FUNCTION TryConvert_REAL_TO_UINT : BOOL
VAR_INPUT
	in : REAL;
	out : REFERENCE TO UINT;
END_VAR

IF in > DatatypeLimits.MAX_VALUE_OF_REAL_WHICH_CAN_BE_HELD_IN_A_UINT THEN
	RETURN;
END_IF

IF in < DatatypeLimits.MIN_VALUE_OF_REAL_WHICH_CAN_BE_HELD_IN_A_UINT THEN
	RETURN;
END_IF

out := REAL_TO_UINT(in);
TryConvert_REAL_TO_UINT := TRUE;

END_FUNCTION

(* stored: Version 1.1.0.1, ProductVersion 3.1.4024.12
   POU TryConvert_REAL_TO_UINT: Id {a0df789c-474f-41b7-af0e-c50eed1a5106}, SpecialFunc None *)
